// TIA Portal V20 export
// export: Created 2025-09-12T17:57:00.0000000Z, ExportSetting WithDefaults
TYPE "UDT300_EM_Heating"
   STRUCT
      HW_Freeze_Stat_DI : Bool;   // Digital Input: Freeze-stat on hot water coil (`True` = Fault).
      HW_Valve_Fdbk_AI : Real;   // Analog Input: Hot water valve position feedback (0-100%).
      HW_Valve_Cmd_AO : Real;   // Analog Output: Hot water valve position command (0-100%).
      HW_Freeze_Alm : Bool;   // Alarm: Hot water coil freeze-stat has tripped.
      Valve_Failure_Alm : Bool;   // Alarm: `True` if valve command and feedback do not match.
   END_STRUCT;
END_TYPE
